ABB RAPID module: CalibData.modx

MODULE CalibData
    PERS tooldata Tooldata_1:=[TRUE,[[0.19321156,0,204.571412367],[0.00026378,0.015111926,-0.999847707,-0.008724874]],[1,[0,0,1],[1,0,0,0],0,0,0]];
    PERS wobjdata Workobject_1:=[FALSE,TRUE,"",[[200.31,-191.81,4.62],[0.999981,0.00480611,-0.00372429,-0.000685934]],[[0,0,0],[1,0,0,0]]];

ENDMODULE
